// TIA Portal V17 export
// export: Created 2023-11-29T12:18:11.2971802Z, ExportSetting WithDefaults, DisplayName Totally Integrated Automation Portal, DisplayVersion V17, DisplayName TIA Portal Openness, DisplayVersion V17, DisplayName TIA Portal Teamcenter Gateway, DisplayVersion V17, DisplayName TIA Portal Version Control Interface, DisplayVersion V17, DisplayName STEP 7 Professional, DisplayVersion V17, DisplayName STEP 7 Safety, DisplayVersion V17, DisplayName WinCC Advanced / Unified PC, DisplayVersion V17
FUNCTION_BLOCK "Baustein_1"   // FB1, FBD
{ S7_Optimized_Access := 'TRUE' }
VERSION : 0.1
// stored: AutoNumber true, IsIECCheckEnabled false, IsRetainMemResEnabled false, MemoryReserve 100, SetENOAutomatically false, UDAEnableTagReadback false
   VAR_OUTPUT
      VarB0 : Bool;
      VarB1 : Bool;
      VarB2 : Bool;
      Varb4 : Bool;
      VarS1 : Bool;
   END_VAR
   VAR_IN_OUT
      Test : Bool;
      Test2 : Bool;
   END_VAR
   VAR_TEMP   // added for the SCL form of the ladder/FBD networks
      _w1 : Bool;
   END_VAR
BEGIN

REGION Network 1
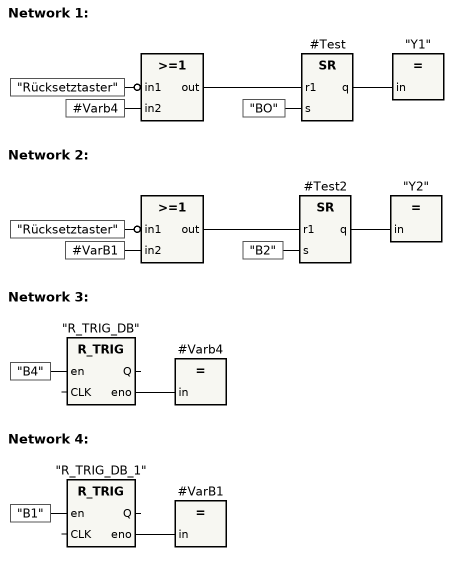
   IF "BO" THEN
       #Test := TRUE;   // SR flip-flop
   END_IF;
   IF NOT "Rücksetztaster" OR #Varb4 THEN #Test := FALSE; END_IF;
   "Y1" := #Test;
END_REGION

REGION Network 2
   IF "B2" THEN
       #Test2 := TRUE;   // SR flip-flop
   END_IF;
   IF NOT "Rücksetztaster" OR #VarB1 THEN #Test2 := FALSE; END_IF;
   "Y2" := #Test2;
END_REGION

REGION Network 3
   "R_TRIG_DB"(EN := "B4", ENO => #_w1);   // R_TRIG
   #Varb4 := #_w1;
END_REGION

REGION Network 4
   "R_TRIG_DB_1"(EN := "B1", ENO => #_w1);   // R_TRIG
   #VarB1 := #_w1;
END_REGION
END_FUNCTION_BLOCK
